(* PLC project Senza_nome, Sconosciuto Senza_nome 1 *)
(* stored: creationDateTime 2021-09-08T11:48:45, modificationDateTime 2021-09-08T14:45:24 *)

FUNCTION function1 : BOOL
  VAR_INPUT
    LOWWORD : UINT;
    HIGHWORD : UINT;
  END_VAR
  VAR_OUTPUT
    WORDSTOREAL : REAL;
  END_VAR

            {{
  union words_to_real {
  uint16_t i[2];
  float f;
  }w2r;
  w2r.i[0] = LOWWORD;
  w2r.i[1] = HIGHWORD;
  WORDSTOREAL = w2r.f;
  }}
          
END_FUNCTION

FUNCTION function2 : BOOL
  VAR_INPUT
    INPUT : REAL;
  END_VAR
  VAR_OUTPUT
    LOWW : UINT;
    HIGG : UINT;
  END_VAR

            {{
  union real_to_words {
  uint16_t i[2];
  float f;
  }r2w;
  r2w.f = INPP;
  LOWW = r2w.i[0];
  HIGG = r2w.i[1];
  }}
          
END_FUNCTION

FUNCTION_BLOCK control
  VAR_INPUT
    PRESSURE : REAL;
    LOAD : REAL;
  END_VAR
  VAR_OUTPUT
    controll : REAL;
  END_VAR

              IF (LOAD = 0.0) THEN
    controll := 1.0;
  ELSIF (PRESSURE<1.015 and LOAD = 1.0) THEN
    controll := 0.0;
  ELSIF (controll = 0.0 and PRESSURE<2.4 and LOAD = 1.0) THEN
    controll := 0.0;
  ELSIF (controll = 0.0 and PRESSURE>2.4 and LOAD = 1.0) THEN
    controll := 1.0;
  ELSIF (controll =1.0 and PRESSURE<2.4 and LOAD = 1.0) THEN
    controll := 1.0;
  END_IF; 
          
END_FUNCTION_BLOCK

PROGRAM plc_actions

(* FBD diagram, written out as Structured Text *)
END_PROGRAM

CONFIGURATION Config0
  RESOURCE Res0 ON PLC
    TASK task0(INTERVAL := T#20ms, PRIORITY := 0);
    PROGRAM instance0 WITH task0 : double_control;
  END_RESOURCE
END_CONFIGURATION
